FUNCTION_BLOCK FB_INPUT_HANDLER
VAR_INPUT
	orgIN : BOOL;
	onlineSwitch : BOOL;
	offLineState : BOOL;
END_VAR
VAR_OUTPUT
	resultIN : BOOL;
	onlineImageID : STRING(20);
 	modeImageID : STRING(20);
END_VAR
VAR
	orgIN_old : BOOL;
	onlineSwitch_old : BOOL;
	offLineState_old : BOOL;
END_VAR

IF GVL.firstCycle THEN
	
	IF onlineSwitch THEN
		onlineImageID := 'switch_on';
		modeImageID := 'switch_undef';
	ELSE
		onlineImageID := 'switch_off';
		
		IF offLineState THEN
			modeImageID := 'switch_on';
		ELSE
			modeImageID := 'switch_off';
		END_IF
		
	END_IF
	
	
	
END_IF

IF onlineSwitch THEN
	resultIN := orgIN;
	IF onlineSwitch <> onlineSwitch_old THEN
		onlineImageID := 'switch_on';
		modeImageID := 'switch_undef';
	END_IF
	
	offLineState := FALSE;
	(* IF offLineState <> offLineState_old THEN
		modeImageID := 'switch_undef';
	END_IF *)
	
ELSE	
	IF onlineSwitch <> onlineSwitch_old THEN
		onlineImageID := 'switch_off';
	END_IF

	IF offLineState THEN
		resultIN := TRUE;
		IF offLineState <> offLineState_old THEN
			modeImageID := 'switch_on';
		END_IF
	ELSE
		resultIN := FALSE;
		IF offLineState <> offLineState_old THEN
			modeImageID := 'switch_off';
		END_IF
	END_IF

END_IF
orgIN_old := orgIN;
onlineSwitch_old := onlineSwitch;
offLineState_old := offLineState;

END_FUNCTION_BLOCK

(* stored: Version 1.1.0.1, ProductVersion 3.1.4024.3
   POU FB_INPUT_HANDLER: Id {077f78e5-6245-4296-932c-8b4771fba0c7}, SpecialFunc None *)
